// TwinCAT 3 PLC project plc01
// ProgramVersion: 3.1.4026.19
// libraries:
//   Tc2_Standard, * (Beckhoff Automation GmbH)
//   Tc2_System, * (Beckhoff Automation GmbH)
//   Tc2_Utilities, * (Beckhoff Automation GmbH)
//   Tc3_EventLogger, * (Beckhoff Automation GmbH)
// project tree:
//   DUTs/ E_LogLevel.TcDUT (not stored), F_Format.TcPOU (not stored), I_Logger.TcIO, I_Logging.TcIO, ST_Message.TcDUT
//   / FastTask.TcTTO (not stored), PlcTask.TcTTO
//   POUs/ FAST.TcPOU, F_InstancePath.TcPOU (not stored), MAIN.TcPOU
//   POUs/FileLogging/ FB_FileLogging.TcPOU
//   POUs/Logger/ FB_Logger.TcPOU
//   POUs/Logging/ FB_Logging.TcPOU
//   POUs/TcLogging/ FB_TcLogging.TcPOU
//   POUs/TcAlarming/ FB_TcAlarming.TcPOU
// real-time tasks:
//   TASK SlowTask: cycle T#20ms, priority 20, ADS port 350
//   TASK FastTask: cycle T#1ms, priority 1, ADS port 351

CONFIGURATION plc01
    RESOURCE PLC ON TwinCAT3
        TASK PlcTask(INTERVAL := T#10ms, PRIORITY := 20);
        PROGRAM MAIN WITH PlcTask : MAIN;
    END_RESOURCE
END_CONFIGURATION

// ---- DUTs/ST_Message.TcDUT
TYPE ST_Message :
STRUCT
	eLogLevel:			E_LogLevel;
	nID:				UDINT;
 	{attribute 'displaymode':='LDT'} 
	nTimestamp:			ULINT;	
	sSource:			STRING(255);
	sMessage:			STRING(255);
	sDefault:			STRING(255);
	sArguments:			STRING(255);
	bActive:			BOOL;
END_STRUCT
END_TYPE

// ---- DUTs/I_Logger.TcIO
INTERFACE I_Logger

METHOD PUBLIC M_AddBOOL
VAR_INPUT
	nValue:				LINT;
END_VAR
END_METHOD

METHOD PUBLIC M_AddINT
VAR_INPUT
	nValue:				LINT;
END_VAR
END_METHOD

METHOD PUBLIC M_AddREAL
VAR_INPUT
	fValue:				LREAL;
	nDecimals:			USINT;
END_VAR
END_METHOD

METHOD PUBLIC M_AddSTRING
VAR_INPUT
	sValue:				STRING(255);
END_VAR
END_METHOD

METHOD PUBLIC M_AddTIME
VAR_INPUT
	tValue:				TIME;
END_VAR
END_METHOD

METHOD PUBLIC M_Debug : BOOL
VAR_INPUT
	sMessage:			STRING(255);
END_VAR
END_METHOD

METHOD PUBLIC M_Error : BOOL
VAR_INPUT
	nID:				UDINT;
	sMessage:			STRING(255);
END_VAR
END_METHOD

METHOD PUBLIC M_Fatal : BOOL
VAR_INPUT
	nID:				UDINT;
	sMessage:			STRING(255);
END_VAR
END_METHOD

METHOD PUBLIC M_Info : BOOL
VAR_INPUT
	nID:				UDINT;
	sMessage:			STRING(255);
END_VAR
END_METHOD

METHOD PUBLIC M_Warn : BOOL
VAR_INPUT
	nID:				UDINT;
	sMessage:			STRING(255);
END_VAR
END_METHOD

END_INTERFACE

// ---- DUTs/I_Logging.TcIO
INTERFACE I_Logging

METHOD PUBLIC M_Attach : BOOL
VAR_INPUT
	iLogging:				I_Logging;
END_VAR
END_METHOD

METHOD PUBLIC M_Log : BOOL
VAR_INPUT
	stMessage:			ST_Message;
END_VAR
END_METHOD

END_INTERFACE

// ---- POUs/MAIN.TcPOU
PROGRAM MAIN
VAR
	fbLogging:			FB_Logging;
	fbTcLogging:		FB_TcLogging;
	fbTcAlarming:		FB_TcAlarming;
	fbLogger:			FB_Logger;
	bVerbose:			BOOL;
	bInfo:				BOOL;
	bWarning:			BOOL;
	bError:				BOOL;
	bCritical:			BOOL;
END_VAR

// toDo 
// * integrate a twincat logger
// * integrate a file logger

fbLogging();
fbLogging.M_Attach(fbTcLogging);

fbTcLogging();

fbTcAlarming();

fbLogger.iLogging:= fbLogging;

fbLogger();

IF bVerbose THEN
	fbLogger.M_AddINT(134052566194980000);
	fbLogger.M_AddSTRING('mm');
	fbLogger.M_Verbose('Verbose message %s %s');
END_IF

IF bInfo THEN
	fbLogger.M_Info(2276475569, 'Info message');
END_IF

IF bWarning THEN
	fbLogger.M_Warning(1791326186, 'Warning message');
END_IF

IF bError THEN
	fbLogger.M_Error(2621541999, 'Error message');
END_IF

IF bCritical THEN
	fbLogger.M_Critical(2626343866, 'Critical message');
END_IF

END_PROGRAM

// ---- POUs/Logging/FB_Logging.TcPOU
// Provide logging 
FUNCTION_BLOCK FB_Logging IMPLEMENTS I_Logging
VAR_INPUT
	eLogLevel:				E_LogLevel:= E_LogLevel.Verbose;
END_VAR
VAR_OUTPUT
    bInfo:					BOOL;
    bWarning:				BOOL;
    bError:					BOOL;
    bCritical:				BOOL;
END_VAR
VAR
	aMessages:				ARRAY[0..99] OF ST_Message; // Message store
    nMessages:				UINT := 0;                     // Message count
	{attribute 'hide'} 
	nIndex: 				UINT;
	iLogging:				I_Logging;
END_VAR

nIndex := 0;
WHILE nIndex < nMessages DO
	IF aMessages[nIndex].bActive THEN
		aMessages[nIndex].bActive:= FALSE;
		nIndex := nIndex + 1;
	ELSE
		IF iLogging <> 0 THEN
			// publish outdated messages to remove
			iLogging.M_Log(aMessages[nIndex]);
		END_IF
        MEMMOVE(ADR(aMessages[nIndex]), ADR(aMessages[nIndex + 1]), SIZEOF(ST_Message) * (nMessages - nIndex));
        nMessages := nMessages - 1;
		bInfo:=	FALSE;
		bWarning:=	FALSE;
		bError:= FALSE;
		bCritical:= FALSE;
    END_IF
END_WHILE

METHOD PUBLIC M_Attach : BOOL
VAR_INPUT
	iLogging:				I_Logging;
END_VAR
IF THIS^.iLogging = 0 THEN
	THIS^.iLogging:= iLogging;
	M_Attach:= TRUE;
ELSIF THIS^.iLogging = iLogging THEN
	// already inside
	M_Attach:= TRUE;
	RETURN;
ELSE
	// redirect to next logging function block
	THIS^.iLogging.M_Attach(iLogging);
END_IF
END_METHOD

METHOD PUBLIC M_Log : BOOL
VAR_INPUT
	stMessage:			ST_Message;
END_VAR
VAR
END_VAR
IF eLogLevel > stMessage.eLogLevel THEN
	M_Log:= TRUE;
	RETURN;
END_IF

CASE stMessage.eLogLevel OF
	E_LogLevel.Info:
    	bInfo:= TRUE;
		
	E_LogLevel.Warning:		
    	bWarning:= TRUE;
		
	E_LogLevel.Error:
    	bError:= TRUE;
		
	E_LogLevel.Critical:
    	bCritical:= TRUE;
		
	ELSE
		;
END_CASE


// Find
FOR nIndex := 0 TO nMessages DO
    IF aMessages[nIndex].sMessage = stMessage.sMessage AND_THEN aMessages[nIndex].sSource = stMessage.sSource THEN
        aMessages[nIndex].bActive:= TRUE;
		M_Log := TRUE;
        RETURN;
    END_IF
END_FOR

// else Add
IF nMessages < 99 THEN
	nIndex := nMessages;
	stMessage.bActive:= TRUE;
    aMessages[nMessages]:= stMessage;;
    nMessages := nMessages + 1;
	// reduce internal buffers 
	// publish new messages to log
	IF iLogging <> 0 THEN
		iLogging.M_Log(stMessage);
	END_IF
	M_Log := TRUE;
END_IF
END_METHOD

PROPERTY PUBLIC P_LogLevel : E_LogLevel
GET
P_LogLevel:= eLogLevel;
END_GET
SET
eLogLevel:= P_LogLevel;
END_SET
END_PROPERTY

END_FUNCTION_BLOCK

// ---- POUs/TcLogging/FB_TcLogging.TcPOU
// Provide logging 
FUNCTION_BLOCK FB_TcLogging IMPLEMENTS I_Logging
VAR_INPUT
	eLogLevel:				E_LogLevel:= E_LogLevel.Verbose;
END_VAR
VAR_OUTPUT
END_VAR
VAR
	iLogging:				I_Logging;
END_VAR

METHOD PUBLIC M_Attach : BOOL
VAR_INPUT
	iLogging:				I_Logging;
END_VAR
IF THIS^.iLogging = 0 THEN
	THIS^.iLogging:= iLogging;
	M_Attach:= TRUE;
ELSIF THIS^.iLogging = iLogging THEN
	// already inside
	M_Attach:= TRUE;
	RETURN;
ELSE
	// redirect to next logging function block
	THIS^.iLogging.M_Attach(iLogging);
END_IF
END_METHOD

METHOD PUBLIC M_Log : BOOL
VAR_INPUT
	stMessage:			ST_Message;
END_VAR
VAR
	fbMsg:				FB_TcMessage; 
	fbSourceInfo:		FB_TcSourceInfo;
END_VAR
IF THIS^.eLogLevel > eLogLevel THEN
	M_Log:= TRUE;
	RETURN;
END_IF

IF stMessage.bActive THEN

	fbSourceInfo.Clear();
	fbSourceInfo.sName:= stMessage.sSource;
	
	CASE stMessage.eLogLevel OF
		E_LogLevel.Verbose:
			fbMsg.CreateEx(TC_EVENTS.TcLogging.Verbose, fbSourceInfo); 	
	
		E_LogLevel.Info:
			fbMsg.CreateEx(TC_EVENTS.TcLogging.Info, fbSourceInfo); 
			
		E_LogLevel.Warning:		
			fbMsg.CreateEx(TC_EVENTS.TcLogging.Warning, fbSourceInfo); 
			
		E_LogLevel.Error:
			fbMsg.CreateEx(TC_EVENTS.TcLogging.Error, fbSourceInfo); 
			
		E_LogLevel.Critical:
			fbMsg.CreateEx(TC_EVENTS.TcLogging.Critical, fbSourceInfo); 
			
	END_CASE
	
	fbMsg.ipArguments.Clear().AddString(stMessage.sDefault);
	
	fbMsg.Send(stMessage.nTimestamp);

END_IF
END_METHOD

PROPERTY PUBLIC P_LogLevel : E_LogLevel
GET
P_LogLevel:= eLogLevel;
END_GET
SET
eLogLevel:= P_LogLevel;
END_SET
END_PROPERTY

END_FUNCTION_BLOCK

// ---- POUs/TcAlarming/FB_TcAlarming.TcPOU
// Provide logging 
FUNCTION_BLOCK FB_TcAlarming IMPLEMENTS I_Logging
VAR_INPUT
	eLogLevel:				E_LogLevel:= E_LogLevel.Verbose;
END_VAR
VAR_OUTPUT
END_VAR
VAR
	iLogging:				I_Logging;
	fbAlarm:				FB_TcAlarm; 
	bInit: BOOL;
END_VAR

IF NOT bInit THEN
	bInit:= TRUE;
	fbAlarm.CreateEx(TC_EVENTS.TcLogging.Verbose, FALSE, 0);
END_IF

IF fbAlarm.bRaised THEN
	;
ELSE
	fbAlarm.Raise(0);
END_IF

//    	fbMsg.CreateEx(TC_EVENTS.TcLogging.Verbose, fbSourceInfo);

METHOD PUBLIC M_Attach : BOOL
VAR_INPUT
	iLogging:				I_Logging;
END_VAR
IF THIS^.iLogging = 0 THEN
	THIS^.iLogging:= iLogging;
	M_Attach:= TRUE;
ELSIF THIS^.iLogging = iLogging THEN
	// already inside
	M_Attach:= TRUE;
	RETURN;
ELSE
	// redirect to next logging function block
	THIS^.iLogging.M_Attach(iLogging);
END_IF
END_METHOD

METHOD PUBLIC M_Log : BOOL
VAR_INPUT
	stMessage:			ST_Message;
END_VAR
VAR
	fbSourceInfo:		FB_TcSourceInfo;
END_VAR
// IF THIS^.eLogLevel > eLogLevel THEN
// 	M_Log:= TRUE;
// 	RETURN;
// END_IF
// 
// fbSourceInfo.Clear();
// fbSourceInfo.sName:= stMessage.sSource;
// 
// CASE eLogLevel OF
// 	E_LogLevel.Verbose:
//     	fbMsg.CreateEx(TC_EVENTS.TcLogging.Verbose, fbSourceInfo); 	
// 
// 	E_LogLevel.Info:
//     	fbMsg.CreateEx(TC_EVENTS.TcLogging.Info, fbSourceInfo); 
// 		
// 	E_LogLevel.Warning:		
//     	fbMsg.CreateEx(TC_EVENTS.TcLogging.Warning, fbSourceInfo); 
// 		
// 	E_LogLevel.Error:
//     	fbMsg.CreateEx(TC_EVENTS.TcLogging.Error, fbSourceInfo); 
// 		
// 	E_LogLevel.Critical:
//     	fbMsg.CreateEx(TC_EVENTS.TcLogging.Critical, fbSourceInfo); 
// 		
// END_CASE
// 
// fbMsg.ipArguments.Clear().AddString(stMessage.sDefault);
// 
// fbMsg.Send(stMessage.nTimestamp);
END_METHOD

PROPERTY PUBLIC P_LogLevel : E_LogLevel
GET
P_LogLevel:= eLogLevel;
END_GET
SET
eLogLevel:= P_LogLevel;
END_SET
END_PROPERTY

END_FUNCTION_BLOCK

// ---- POUs/Logger/FB_Logger.TcPOU
{attribute 'reflection'} 
FUNCTION_BLOCK FB_Logger
VAR_INPUT
	iLogging:			I_Logging;
END_VAR
VAR_OUTPUT
END_VAR
VAR
    {attribute 'instance-path'} 
    {attribute 'noinit'} 
    sInstancePath:				STRING(255); 
	sArguments:					STRING(255); 
END_VAR

//FB_Init ist immer implizit verfügbar und wird primär für die Initialisierung verwendet.
//Der Rückgabewert wird nicht ausgewertet. Für gezielte Einflussnahme können Sie
//die Methoden explizit deklarieren und darin mit dem Standard-Initialisierungscode 
//zusätzlichen Code bereitstellen. Sie können den Rückgabewert auswerten.
METHOD FB_Init: BOOL
VAR_INPUT    
bInitRetains: BOOL; // TRUE: Die Retain-Variablen werden initialisiert (Reset warm / Reset kalt)    
bInCopyCode: BOOL;  // TRUE: Die Instanz wird danach in den Kopiercode kopiert (Online-Change)
END_VAR
sInstancePath:= F_InstancePath(sInstancePath);
END_METHOD

METHOD PUBLIC M_AddBOOL
VAR_INPUT
	nValue:				LINT;
END_VAR
VAR
	sValue: 			STRING;
END_VAR
sValue:= LINT_TO_STRING(nValue);			// convert
sValue:= CONCAT(sValue, '$R');				// add separator
sArguments:= CONCAT(sArguments, sValue);	// add new arg
END_METHOD

METHOD PUBLIC M_AddINT
VAR_INPUT
	nValue:				LINT;
END_VAR
VAR
	sValue: 			STRING;
END_VAR
sValue:= LINT_TO_STRING(nValue);			// convert
sValue:= CONCAT(sValue, '$R');				// add separator
sArguments:= CONCAT(sArguments, sValue);	// add new arg
END_METHOD

METHOD PUBLIC M_AddREAL
VAR_INPUT
	fValue:				LREAL;
	nDecimals:			USINT;
END_VAR
VAR
	sValue: 			STRING;
END_VAR
sValue:= LREAL_TO_FMTSTR(fValue, nDecimals, TRUE);		// convert
sValue:= CONCAT(sValue, '$R');							// add separator
sArguments:= CONCAT(sArguments, sValue);				// add new arg
END_METHOD

METHOD PUBLIC M_AddSTRING
VAR_INPUT
	sValue:				STRING(255);
END_VAR
sValue:= CONCAT(sValue, '$R');				// add separator
sArguments:= CONCAT(sArguments, sValue);	// add new arg
END_METHOD

METHOD PUBLIC M_AddTIME
VAR_INPUT
	tValue:				TIME;
END_VAR
VAR
	sValue: 			STRING;
END_VAR
sValue:= TIME_TO_STRING(tValue);			// convert
sValue:= CONCAT(sValue, '$R');				// add separator
sArguments:= CONCAT(sArguments, sValue);	// add new arg
END_METHOD

METHOD PUBLIC M_Critical : BOOL
VAR_INPUT
	nID:				UDINT;
	sMessage:			STRING(255);
END_VAR
VAR
	stMessage:			ST_Message;
END_VAR
IF iLogging = 0 THEN
	RETURN;
END_IF

stMessage.eLogLevel:= E_LogLevel.Critical;
stMessage.nID:= nID;
stMessage.nTimestamp:= F_GetSystemTime();
stMessage.sMessage:= sMessage;
stMessage.sArguments:= sArguments;
stMessage.sDefault:= F_Format(sMessage, sArguments);
stMessage.sSource:= sInstancePath;
sArguments:= '';

iLogging.M_Log(stMessage);
END_METHOD

METHOD PUBLIC M_Error : BOOL
VAR_INPUT
	nID:				UDINT;
	sMessage:			STRING(255);
END_VAR
VAR
	stMessage:			ST_Message;
END_VAR
IF iLogging = 0 THEN
	RETURN;
END_IF

stMessage.eLogLevel:= E_LogLevel.Error;
stMessage.nID:= nID;
stMessage.nTimestamp:= F_GetSystemTime();
stMessage.sMessage:= sMessage;
stMessage.sArguments:= sArguments;
stMessage.sDefault:= F_Format(sMessage, sArguments);
stMessage.sSource:= sInstancePath;
sArguments:= '';

iLogging.M_Log(stMessage);
END_METHOD

METHOD PUBLIC M_Info : BOOL
VAR_INPUT
	nID:				UDINT;
	sMessage:			STRING(255);
END_VAR
VAR
	stMessage:			ST_Message;
END_VAR
IF iLogging = 0 THEN
	RETURN;
END_IF

stMessage.eLogLevel:= E_LogLevel.Info;
stMessage.nID:= nID;
stMessage.nTimestamp:= F_GetSystemTime();
stMessage.sMessage:= sMessage;
stMessage.sArguments:= sArguments;
stMessage.sDefault:= F_Format(sMessage, sArguments);
stMessage.sSource:= sInstancePath;
sArguments:= '';

iLogging.M_Log(stMessage);
END_METHOD

METHOD PUBLIC M_Verbose : BOOL
VAR_INPUT
	sMessage:			STRING(255);
END_VAR
VAR
	stMessage:			ST_Message;
END_VAR
IF iLogging = 0 THEN
	RETURN;
END_IF

stMessage.eLogLevel:= E_LogLevel.Verbose;
stMessage.nID:= 0;
stMessage.nTimestamp:= F_GetSystemTime();
stMessage.sMessage:= sMessage;
stMessage.sArguments:= sArguments;
stMessage.sDefault:= F_Format(sMessage, sArguments);
stMessage.sSource:= sInstancePath;
sArguments:= '';

iLogging.M_Log(stMessage);
END_METHOD

METHOD PUBLIC M_Warning : BOOL
VAR_INPUT
	nID:				UDINT;
	sMessage:			STRING(255);
END_VAR
VAR
	stMessage:			ST_Message;
END_VAR
IF iLogging = 0 THEN
	RETURN;
END_IF

stMessage.eLogLevel:= E_LogLevel.Warning;
stMessage.nID:= nID;
stMessage.nTimestamp:= F_GetSystemTime();
stMessage.sMessage:= sMessage;
stMessage.sArguments:= sArguments;
stMessage.sDefault:= F_Format(sMessage, sArguments);
stMessage.sSource:= sInstancePath;
sArguments:= '';

iLogging.M_Log(stMessage);
END_METHOD

PROPERTY PUBLIC P_Logger : I_Logging
GET
P_Logger:= iLogging;
END_GET
SET
iLogging:= P_Logger;
END_SET
END_PROPERTY

END_FUNCTION_BLOCK

// ---- POUs/FAST.TcPOU
PROGRAM FAST
VAR
	fbLogger:			FB_Logger;
	bVerbose:			BOOL;
	bInfo:				BOOL;
	bWarning:			BOOL;
	bError:				BOOL;
	bCritical:			BOOL;
END_VAR

fbLogger.P_Logger:= MAIN.fbLogging;

IF bVerbose THEN
	fbLogger.M_AddINT(134052566194980000);
	fbLogger.M_AddSTRING('mm');
	fbLogger.M_Verbose('Verbose message %s %s');
END_IF

IF bInfo THEN
	fbLogger.M_Info(2276475569, 'Info message');END_IF

IF bWarning THEN
	fbLogger.M_Info(2276475569, 'Info message');
	fbLogger.M_Info(2276475569, 'Info message');
	fbLogger.M_Warning(1791326186, 'Warning message');
	fbLogger.M_Error(2621541999, 'Error message');
END_IF

IF bError THEN

END_IF

IF bCritical THEN
	fbLogger.M_Critical(2626343866, 'Critical message');
END_IF

END_PROGRAM

// ---- POUs/FileLogging/FB_FileLogging.TcPOU
// Provide logging 
FUNCTION_BLOCK FB_FileLogging IMPLEMENTS I_Logging
VAR_INPUT
	eLogLevel:				E_LogLevel:= E_LogLevel.Verbose;
END_VAR
VAR_OUTPUT
END_VAR
VAR
	iLogging:				I_Logging;
END_VAR

METHOD PUBLIC M_Attach : BOOL
VAR_INPUT
	iLogging:				I_Logging;
END_VAR
IF THIS^.iLogging = 0 THEN
	THIS^.iLogging:= iLogging;
	M_Attach:= TRUE;
ELSIF THIS^.iLogging = iLogging THEN
	// already inside
	M_Attach:= TRUE;
	RETURN;
ELSE
	// redirect to next logging function block
	THIS^.iLogging.M_Attach(iLogging);
END_IF
END_METHOD

METHOD PUBLIC M_Log : BOOL
VAR_INPUT
	eLogLevel:			E_LogLevel;
	nID:				UDINT;
	sSource:			STRING(255);
	sMessage:			STRING(255);
	sArguments:			STRING(255);
END_VAR
VAR
	fbMsg:				FB_TcLogging; 
	fbSourceInfo:		FB_TcSourceInfo;
END_VAR
END_METHOD

PROPERTY PUBLIC P_LogLevel : E_LogLevel
GET
P_LogLevel:= eLogLevel;
END_GET
SET
eLogLevel:= P_LogLevel;
END_SET
END_PROPERTY

END_FUNCTION_BLOCK
